INTERFACE I_Nasmyth

METHOD SetNasmyth : BOOL
VAR_INPUT
	Port	: USINT;
END_VAR
END_METHOD

END_INTERFACE

(* stored: Version 1.1.0.1, ProductVersion 3.1.4024.13
   POU I_Nasmyth: Id {4813c151-6664-41fc-a0d0-2e76bd1bea8d}, SpecialFunc None
   Method SetNasmyth: Id {e1c0b1d1-b238-4570-9066-517811e0b058} *)
